// TIA Portal V20 export
// export: Created 2025-12-01T14:57:04.1279585Z, ExportSetting None, DisplayName Totally Integrated Automation Portal, DisplayVersion V20 Update 3, DisplayName TIA Portal Openness, DisplayVersion V20 Update 3, DisplayName TIA Portal Version Control Interface, DisplayVersion V20 Update 3, DisplayName STEP 7 Professional, DisplayVersion V20 Update 3, DisplayName STEP 7 Safety, DisplayVersion V20 Update 2, DisplayName WinCC Basic/Comfort/Advanced, DisplayVersion V20 Update 3, DisplayName WinCC Professional, DisplayVersion V20 Update 3, DisplayName WinCC Unified, DisplayVersion V20 Update 3
FUNCTION "FC706_JDT02Borrado" : Void   // FC706, LAD
TITLE = "BorrodoTracking" - Borrado de toda la Base de Datos
{ S7_Optimized_Access := 'FALSE' }
AUTHOR : TRACKING
NAME : 20130301
VERSION : 3.0
// - Borrado de todos los DB's
// - Inicializadcion del DB de DatosUT
// stored: AutoNumber false, SetENOAutomatically false
   VAR_TEMP
      NumeroUT : Int;
      NumDB : Word;
      UTVacia : Int;
   END_VAR
BEGIN

NETWORK
TITLE = Borrado de todos los DB's de Comunicacion
// -------------------------------------------------------------------------------
// --- Mirar si hay que resetear
      AN    "DB701_JDT02StatusCOM".ResetBD;
      JC    NoResetear;

// -------------------------------------------------------------------------------
// Borrado de los DB de Recepcion de Eventos

      CALL  "FC898_BorrarMensaje"
      ( DB_A_RESET := "DB702_JDT02RecepMensaje"
      );
      CALL  "FC898_BorrarMensaje"
      ( DB_A_RESET := "DB704_JDT02UltimoRecibido"
      );
      CALL  "FC898_BorrarMensaje"
      ( DB_A_RESET := "DB708_JDT02EventosRecibidos"
      );

// -------------------------------------------------------------------------------
// Borrado de los DB de Emision de Eventos

      CALL  "FC898_BorrarMensaje"
      ( DB_A_RESET := "DB703_JDT02EmisionMensaje"
      );
      CALL  "FC898_BorrarMensaje"
      ( DB_A_RESET := "DB705_JDT02UltimoEnviado"
      );
      CALL  "FC898_BorrarMensaje"
      ( DB_A_RESET := "DB706_JDT02EmisionAK"
      );
      CALL  "FC898_BorrarMensaje"
      ( DB_A_RESET := "DB707_JDT02EventosGenerados"
      );

// -------------------------------------------------------------------------------
// Borrado de los DB de la BD de Mesas
// El DB de CrucesMesas no se borra, esto es fijo para cada instalación

      CALL  "FC898_BorrarMensaje"
      ( DB_A_RESET := "DB810_ColasMesas"
      );
      CALL  "FC898_BorrarMensaje"
      ( DB_A_RESET := "DB811_ColasMckeys"
      );

      CALL  "FC898_BorrarMensaje"
      ( DB_A_RESET := "DB812_UTs_Control"
      );
      CALL  "FC898_BorrarMensaje"
      ( DB_A_RESET := "DB813_UTs_Ruta"
      );

      CALL  "FC898_BorrarMensaje"
      ( DB_A_RESET := "DB814_UTs_Etiqueta"
      );
      CALL  "FC898_BorrarMensaje"
      ( DB_A_RESET := "DB815_UTs_Datos"
      );
      CALL  "FC898_BorrarMensaje"
      ( DB_A_RESET := "DB816_UTs_TextoPantalla"
      );
      CALL  "FC898_BorrarMensaje"
      ( DB_A_RESET := "DB820_UTs_DatosQUBIQA"
      );
      CALL  "FC898_BorrarMensaje"
      ( DB_A_RESET := "DB821_UTs_DatosIKPAL"
      );


// -------------------------------------------------------------------------------
// Borrado de los DB de la BD de Dispositivos

      CALL  "FC898_BorrarMensaje"
      ( DB_A_RESET := "DB830_Dispositivos"
      );
      CALL  "FC898_BorrarMensaje"
      ( DB_A_RESET := "DB831_Mesas"
      );
      CALL  "FC898_BorrarMensaje"
      ( DB_A_RESET := "DB832_Maquinas"
      );


// -------------------------------------------------------------------------------
// Borrado de los DB Emision y Recepcion con la instalación

      CALL  "FC898_BorrarMensaje"
      ( DB_A_RESET := "DB840_Emision"
      );
      CALL  "FC898_BorrarMensaje"
      ( DB_A_RESET := "DB841_Recepcion"
      );
      CALL  "FC898_BorrarMensaje"
      ( DB_A_RESET := "DB843_RecepcionPantalla"
      );

      SET;
      R     "DB701_JDT02StatusCOM".ResetBD;

      JU    FinFuncion;  // El siguiente segmento no se realiza


NETWORK
TITLE = ----
// Se acabo la inicializacion
NoResetear:NOP   0;
      L     0;
      LAR1;

// -------------------------------------------------------------------------------
// Borrado de los DB de Recepcion de Eventos, si es necesario

      OPN   "DB702_JDT02RecepMensaje";
      L     DBB [AR1, P#0.0];
      L     ' ';
      <>I;
      JC    S_31;
      CALL  "FC898_BorrarMensaje"
      ( DB_A_RESET := "DB702_JDT02RecepMensaje"
      );

S_31: OPN   "DB704_JDT02UltimoRecibido";
      L     DBB [AR1, P#0.0];
      L     ' ';
      <>I;
      JC    S_32;
      CALL  "FC898_BorrarMensaje"
      ( DB_A_RESET := "DB704_JDT02UltimoRecibido"
      );

S_32: OPN   "DB708_JDT02EventosRecibidos";
      L     DBB [AR1, P#0.0];

      L     ' ';
      <>I;
      JC    S_33;
      CALL  "FC898_BorrarMensaje"
      ( DB_A_RESET := "DB708_JDT02EventosRecibidos"
      );

// -------------------------------------------------------------------------------
// Borrado de los DB de Emision de Eventos, si es necesario

S_33: OPN   "DB703_JDT02EmisionMensaje";
      L     DBB [AR1, P#0.0];
      L     ' ';
      <>I;
      JC    S_34;
      CALL  "FC898_BorrarMensaje"
      ( DB_A_RESET := "DB703_JDT02EmisionMensaje"
      );

S_34: OPN   "DB705_JDT02UltimoEnviado";
      L     DBB [AR1, P#0.0];
      L     ' ';
      <>I;
      JC    S_35;
      CALL  "FC898_BorrarMensaje"
      ( DB_A_RESET := "DB705_JDT02UltimoEnviado"
      );

S_35: OPN   "DB706_JDT02EmisionAK";
      L     DBB [AR1, P#0.0];
      L     ' ';
      <>I;
      JC    S_36;
      CALL  "FC898_BorrarMensaje"
      ( DB_A_RESET := "DB706_JDT02EmisionAK"
      );

S_36: OPN   "DB707_JDT02EventosGenerados";
      L     DBB [AR1, P#0.0];
      L     ' ';
      <>I;
      JC    S_39;
      CALL  "FC898_BorrarMensaje"
      ( DB_A_RESET := "DB707_JDT02EventosGenerados"
      );

S_39: NOP   0;
      JU    FinFuncion;


NETWORK
TITLE = Final de la funcion
FinFuncion:NOP   0;



END_FUNCTION
